// Mitsubishi GX Works2 project: 모터6   PLC: Q02/Q02H

PROGRAM MAIN
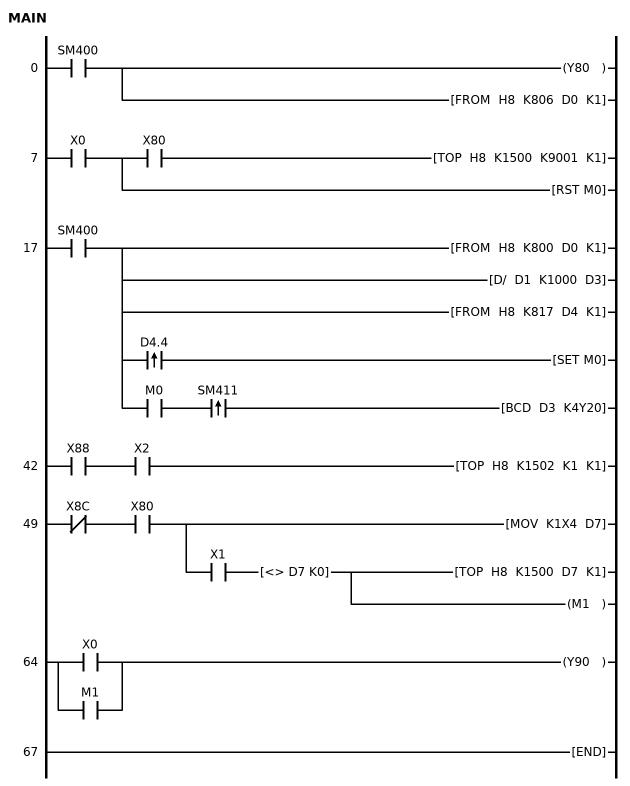
0     LD      SM400
      OUT     Y80
      FROM    H8 K806 D0 K1
7     LD      X0
      MPS
      AND     X80
      TOP     H8 K1500 K9001 K1
      MPP
      RST     M0
17    LD      SM400
      FROM    H8 K800 D0 K1
      D/      D1 K1000 D3
      FROM    H8 K817 D4 K1
      MPS
      ANDP    D4.4
      SET     M0
      MPP
      AND     M0
      ANDP    SM411
      BCD     D3 K4Y20
42    LD      X88
      AND     X2
      TOP     H8 K1502 K1 K1
49    LDI     X8C
      AND     X80
      MOV     K1X4 D7
      AND     X1
      AND<>   D7 K0
      TOP     H8 K1500 D7 K1
      OUT     M1
64    LD      X0
      OR      M1
      OUT     Y90
67    END
END_PROGRAM
